// TIA Portal V20 export
DATA_BLOCK "SBK13"   // DB297
// stored: MemoryReserve 100
   VAR
      "X1-1 SAFETY DOOR LOCK13.INPUT" : Bool;
      "X2-1 SPARE" : Bool;
      "X3-1 SPARE" : Bool;
      "X4-1 SPARE" : Bool;
      "X1-2 SAFETY DOOR LOCK13.INPUT" : Bool;
      "X2-2 SPARE" : Bool;
      "X3-2 SPARE" : Bool;
      "X4-2 SPARE" : Bool;
   END_VAR
BEGIN
END_DATA_BLOCK
